// TIA Portal V17 export
// export: Created 2025-06-25T13:13:29.0172389Z, ExportSetting WithDefaults, DisplayName Totally Integrated Automation Portal, DisplayVersion V17 Update 8, DisplayName TIA Portal Openness, DisplayVersion V17 Update 8, DisplayName TIA Portal Version Control Interface, DisplayVersion V17, DisplayName STEP 7 Professional, DisplayVersion V17 Update 8, DisplayName STEP 7 Safety, DisplayVersion V17 Update 6, DisplayName WinCC Advanced, DisplayVersion V17 Update 8
TYPE "stSM531_8AI"
// stored: IsFailsafeCompliant false
   STRUCT
      CH00 : Int;
      CH01 : Int;
      CH02 : Int;
      CH03 : Int;
      CH04 : Int;
      CH05 : Int;
      CH06 : Int;
      CH07 : Int;
      CH00_ok : Bool;
      CH01_ok : Bool;
      CH02_ok : Bool;
      CH03_ok : Bool;
      CH04_ok : Bool;
      CH05_ok : Bool;
      CH06_ok : Bool;
      CH07_ok : Bool;
   END_STRUCT;
END_TYPE
